Universal Robots PolyScope program: HumanReadableForm.urp

Program rtde_control_loop (createdIn=3.2.19275.0 lastSavedIn=3.6.1.30595 robotSerialNumber=2014359999 directory=/home/ur/ursim-current/programs installation=default)
BeforeStart
  setp := 
  Script: 
  Script: 
Robot Program (runOnlyOnce=false motionType=MoveJ speed=1.047198 acceleration=1.396263 useActiveTCP=false)
  If 
    MoveL speed 80 mm/s, acceleration 1200 mm/s^2 (useActiveTCP=false) feature=Base
      Waypoint Waypoint (Variable): variable=setp
    Script: 
    Loop While (checkContinuously=false)
      Script: 
    Script: 
  Script: 
Thread Thread_1 (runOnlyOnce=false trackProgramExecution=false)
  Loop Forever
    tmp := 
    Script: 
    Script: 
